{attribute 'GeneratedUsingTerminal: AT2020-0250-0019'}
{attribute addProperty BoxType "AT2020-0250-0019"}
{attribute addProperty Id "StatusAT %I*UINT2Current_actual_value_ChAT %I*ARRAY[0..14] OF INT30"}
{attribute addProperty CRC "4120755276"}
{attribute addProperty Size "32"}
TYPE CC_Inputs_2C1C9EE0 EXTENDS InputBase_8311D824 :
STRUCT
	{attribute addProperty Name "Status"}
	Status AT %I* : UINT;
	{attribute addProperty Name "Current_actual_value_Ch"}
	Current_actual_value_Ch AT %I* : ARRAY[0..14] OF INT;
END_STRUCT
END_TYPE

(* stored: Version 1.2.0.0, ProductVersion 3.1.4024.9
   DUT CC_Inputs_2C1C9EE0: Id {a19597b2-e52a-40b4-8d57-4ccaa3779cda} *)
